INTERFACE ITF_BA_Scara

METHOD MC_ChangeSpeedOverride : INT
VAR_INPUT
	factor: REAL;
END_VAR
END_METHOD

METHOD MC_MoveAxesAbsolute : BOOL
VAR_INPUT
	target: stTarget3D;
END_VAR
END_METHOD

METHOD MC_MoveAxesRelative : BOOL
VAR_INPUT
	axes: ARRAY[1..6] OF FB_Axis;
	offsets: ARRAY[1..6] OF REAL;
END_VAR
END_METHOD

METHOD MC_MoveLinearAbsolute : BOOL
VAR_INPUT
	target: stTarget3D;
END_VAR
END_METHOD

METHOD PUBLIC MC_ReadAnalogInput : LREAL
VAR_INPUT
	input : INT;
END_VAR
END_METHOD

METHOD PUBLIC MC_ReadDigitalInput : BOOL
VAR_INPUT
	input : INT;
END_VAR
END_METHOD

METHOD PUBLIC MC_SetDigitalOutput : BOOL
VAR_INPUT
	output : INT;
	value : BOOL;
END_VAR
END_METHOD

METHOD PUBLIC MC_SetOperationMode : BOOL
VAR_INPUT
	mode: eMode;
END_VAR
END_METHOD

END_INTERFACE

(* stored: Version 1.1.0.1, ProductVersion 3.1.4026.18
   Itf ITF_BA_Scara: Id {a1d9ae2a-6d58-4f24-bdfc-a2fb51ab02f5}
   Method MC_ChangeSpeedOverride: Id {34c834d8-9901-43a3-ae1a-8f458d200544}
   Method MC_MoveAxesAbsolute: Id {b14ca16d-ff7d-4202-bcc9-3733bf0888ca}
   Method MC_MoveAxesRelative: Id {b4b961e8-30c8-4602-8978-3235cc9c3d90}
   Method MC_MoveLinearAbsolute: Id {6779f5f0-07a0-4df1-b286-b2c7242ed92e}
   Method MC_ReadAnalogInput: Id {d0798ec4-b248-41b2-ab96-c8b712f3f2fc}
   Method MC_ReadDigitalInput: Id {0e60299c-811b-4dd0-91a7-cf91ee677ae0}
   Method MC_SetDigitalOutput: Id {e0e0d204-e7a4-47f4-84a7-e460e4338a02}
   Method MC_SetOperationMode: Id {6e7ec3fc-b084-4266-a09f-fa2470f60bc8} *)
